Fanuc KAREL source: SEMA_COUNT.kl

PROGRAM T
%NOLOCKGROUP
VAR
 v0 : INTEGER
 res : INTEGER
BEGIN
 res = SEMA_COUNT(v0)
END T
